(* IEC 61131-3 sources: volt/packages/volt-lsp-iec/test-corpus/lenze-mid/Device/Plc Logic/Application/Library Manager/CAA DTUtility, 19 files *)

(* ---- DTU_GETDATEANDTIME_PARAMS.dut ---- *)
TYPE DTU_GETDATEANDTIME_PARAMS :
STRUCT
	DTDATEANDTIME : DATE_AND_TIME;
	ETIMEZONE : RTCLK.PERIODE;
END_STRUCT
END_TYPE

(* ---- DTU_GETTIMEZONEINFORMATION_PARAMS.dut ---- *)
TYPE DTU_GETTIMEZONEINFORMATION_PARAMS :
STRUCT
	TZITIMEZONE : RTCLK.TIME_ZONE_INFO;
END_STRUCT
END_TYPE

(* ---- DTU_SETDATEANDTIME_PARAMS.dut ---- *)
TYPE DTU_SETDATEANDTIME_PARAMS :
STRUCT
	DTDATEANDTIME : DATE_AND_TIME;
END_STRUCT
END_TYPE

(* ---- DTU_SETTIMEZONEINFORMATION_PARAMS.dut ---- *)
TYPE DTU_SETTIMEZONEINFORMATION_PARAMS :
STRUCT
	TZITIMEZONE : RTCLK.TIME_ZONE_INFO;
END_STRUCT
END_TYPE

(* ---- ERROR.dut ---- *)
TYPE ERROR :
(
	NO_ERROR := 0,
	FIRST_ERROR := 5750,
	TIME_OUT := 5751,
	NOT_AVAILABLE := 5752,
	INPUT_INVALID := 5753,
	DTU_ERROR_UNKNOWN := 5754,
	DTU_WRONG_PARAMETER := 5755,
	DTU_TZI_NOT_SET := 5756,
	FIRST_MF := 5770,
	LAST_ERROR := 5799
);
END_TYPE

(* ---- GLOBALCONSTANTS.gvl ---- *)
VAR_GLOBAL
	GC_TZITIMEZONECET : RTCLK.TIME_ZONE_INFO := STRUCT(iBias := 60, sPeriode := [STRUCT(sName := 'CET', tmDate := STRUCT(uiMonth := 10, eWeekday := RTCLK.WEEKDAY.SUNDAY, uiDay := 5, uiHour := 3, uiMinute := 0, uiSecond := 0), iBias := 0), STRUCT(sName := 'CEST', tmDate := STRUCT(uiMonth := 3, eWeekday := RTCLK.WEEKDAY.SUNDAY, uiDay := 5, uiHour := 2, uiMinute := 0, uiSecond := 0), iBias := 60)]);
END_VAR

(* ---- VERSIONCONSTANTS.gvl ---- *)
VAR_GLOBAL
	GC_BYVERSION : BYTE := 1;
	GC_VERSION_1 : BYTE := 0;
END_VAR

(* ---- DATECONCAT.pou ---- *)
FUNCTION DATECONCAT : DATE
VAR_INPUT
	UIYEAR : UINT;
	UIMONTH : UINT;
	UIDAY : UINT;
	PEERROR : POINTER TO ERROR;
END_VAR
END_FUNCTION

(* ---- DATESPLIT.pou ---- *)
FUNCTION DATESPLIT : ERROR
VAR_INPUT
	DATDATE : DATE;
	PUIYEAR : POINTER TO UINT;
	PUIMONTH : POINTER TO UINT;
	PUIDAY : POINTER TO UINT;
END_VAR
END_FUNCTION

(* ---- DTCONCAT.pou ---- *)
FUNCTION DTCONCAT : DATE_AND_TIME
VAR_INPUT
	UIYEAR : UINT;
	UIMONTH : UINT;
	UIDAY : UINT;
	UIHOUR : UINT;
	UIMINUTE : UINT;
	UISECOND : UINT;
	PEERROR : POINTER TO ERROR;
END_VAR
END_FUNCTION

(* ---- DTSPLIT.pou ---- *)
FUNCTION DTSPLIT : ERROR
VAR_INPUT
	DTDATEANDTIME : DATE_AND_TIME;
	PUIYEAR : POINTER TO UINT;
	PUIMONTH : POINTER TO UINT;
	PUIDAY : POINTER TO UINT;
	PUIHOUR : POINTER TO UINT;
	PUIMINUTE : POINTER TO UINT;
	PUISECOND : POINTER TO UINT;
END_VAR
END_FUNCTION

(* ---- GETDAYOFWEEK.pou ---- *)
FUNCTION GETDAYOFWEEK : RTCLK.WEEKDAY
VAR_INPUT
	DTDATE : DATE;
	PEERROR : POINTER TO ERROR;
END_VAR
END_FUNCTION

(* ---- GETSUPPLIERVERSION.pou ---- *)
FUNCTION GETSUPPLIERVERSION : WORD
VAR_INPUT
	XDUMMY : BOOL;
END_VAR
END_FUNCTION

(* ---- TODCONCAT.pou ---- *)
FUNCTION TODCONCAT : TIME_OF_DAY
VAR_INPUT
	UIHOUR : UINT;
	UIMINUTE : UINT;
	UISECOND : UINT;
	UIMILLISECOND : UINT;
	PEERROR : POINTER TO ERROR;
END_VAR
END_FUNCTION

(* ---- TODSPLIT.pou ---- *)
FUNCTION TODSPLIT : ERROR
VAR_INPUT
	TODTIME : TIME_OF_DAY;
	PUIHOUR : POINTER TO UINT;
	PUIMINUTE : POINTER TO UINT;
	PUISECOND : POINTER TO UINT;
	PUIMILLISECOND : POINTER TO UINT;
END_VAR
END_FUNCTION

(* ---- GETDATEANDTIME.pou ---- *)
FUNCTION_BLOCK GETDATEANDTIME
VAR_INPUT
	XEXECUTE : BOOL;
END_VAR
VAR_OUTPUT
	XDONE : BOOL;
	XBUSY : BOOL;
	XERROR : BOOL;
	EERROR : ERROR;
	DTDATEANDTIME : DATE_AND_TIME;
	EPERIODE : RTCLK.PERIODE;
END_VAR
VAR
	XPREVIOUSEXECUTE : BOOL;
	XPREVIOUSABORTINPROGRESS : BOOL;
	XABORTINPROGRESS : BOOL;
	IERROR : INT;
	HJOB : CAA.HANDLE;
	PGETDATEANDTIMEPARAMS : POINTER TO DTU_GETDATEANDTIME_PARAMS;
	STATEJOB : ASM.STATE;
	DWETRIGCLASS : __XWORD;
END_VAR
END_FUNCTION_BLOCK

METHOD FB_INIT : BOOL
VAR_INPUT
	BINITRETAINS : BOOL;
	BINCOPYCODE : BOOL;
END_VAR
END_METHOD

METHOD FB_EXIT : BOOL
VAR_INPUT
	BINCOPYCODE : BOOL;
END_VAR
END_METHOD

(* ---- GETTIMEZONEINFORMATION.pou ---- *)
FUNCTION_BLOCK GETTIMEZONEINFORMATION
VAR_INPUT
	XEXECUTE : BOOL;
END_VAR
VAR_OUTPUT
	XDONE : BOOL;
	XBUSY : BOOL;
	XERROR : BOOL;
	EERROR : ERROR;
	TZIINFO : RTCLK.TIME_ZONE_INFO;
END_VAR
VAR
	XPREVIOUSEXECUTE : BOOL;
	XPREVIOUSABORTINPROGRESS : BOOL;
	XABORTINPROGRESS : BOOL;
	IERROR : INT;
	HJOB : CAA.HANDLE;
	PGETTIMEZONEINFORMATIONPARAMS : POINTER TO DTU_GETTIMEZONEINFORMATION_PARAMS;
	STATEJOB : ASM.STATE;
	DWETRIGCLASS : __XWORD;
END_VAR
END_FUNCTION_BLOCK

METHOD FB_EXIT : BOOL
VAR_INPUT
	BINCOPYCODE : BOOL;
END_VAR
END_METHOD

METHOD FB_INIT : BOOL
VAR_INPUT
	BINITRETAINS : BOOL;
	BINCOPYCODE : BOOL;
END_VAR
END_METHOD

(* ---- SETDATEANDTIME.pou ---- *)
FUNCTION_BLOCK SETDATEANDTIME
VAR_INPUT
	XEXECUTE : BOOL;
	DTDATEANDTIME : DATE_AND_TIME;
END_VAR
VAR_OUTPUT
	XDONE : BOOL;
	XBUSY : BOOL;
	XERROR : BOOL;
	EERROR : ERROR;
END_VAR
VAR
	XPREVIOUSEXECUTE : BOOL;
	XPREVIOUSABORTINPROGRESS : BOOL;
	XABORTINPROGRESS : BOOL;
	IERROR : INT;
	HJOB : CAA.HANDLE;
	PSETDATEANDTIMEPARAMS : POINTER TO DTU_SETDATEANDTIME_PARAMS;
	STATEJOB : ASM.STATE;
	DWETRIGCLASS : __XWORD;
END_VAR
END_FUNCTION_BLOCK

METHOD FB_INIT : BOOL
VAR_INPUT
	BINITRETAINS : BOOL;
	BINCOPYCODE : BOOL;
END_VAR
END_METHOD

METHOD FB_EXIT : BOOL
VAR_INPUT
	BINCOPYCODE : BOOL;
END_VAR
END_METHOD

(* ---- SETTIMEZONEINFORMATION.pou ---- *)
FUNCTION_BLOCK SETTIMEZONEINFORMATION
VAR_INPUT
	XEXECUTE : BOOL;
	TZIINFO : RTCLK.TIME_ZONE_INFO;
END_VAR
VAR_OUTPUT
	XDONE : BOOL;
	XBUSY : BOOL;
	XERROR : BOOL;
	EERROR : ERROR;
END_VAR
VAR
	XPREVIOUSEXECUTE : BOOL;
	XPREVIOUSABORTINPROGRESS : BOOL;
	XABORTINPROGRESS : BOOL;
	IERROR : INT;
	HJOB : CAA.HANDLE;
	PSETTIMEZONEINFORMATIONPARAMS : POINTER TO DTU_SETTIMEZONEINFORMATION_PARAMS;
	STATEJOB : ASM.STATE;
	DWETRIGCLASS : __XWORD;
END_VAR
END_FUNCTION_BLOCK

METHOD FB_INIT : BOOL
VAR_INPUT
	BINITRETAINS : BOOL;
	BINCOPYCODE : BOOL;
END_VAR
END_METHOD

METHOD FB_EXIT : BOOL
VAR_INPUT
	BINCOPYCODE : BOOL;
END_VAR
END_METHOD
